// TIA Portal V20 export
FUNCTION "CollectAlarms" : Void   // FC61, LAD
TITLE = U1Em1_SepaUnwinderBottom
// stored: Namespace Unit1.Em1, SetENOAutomatically false
   VAR_INPUT
      resetAlarms : Bool;
      disableAlarms : Bool;
   END_VAR
   VAR_OUTPUT
      commandsToUnit : "LUC_typeStateCommands";   // Feedback to the unit
   END_VAR
   VAR CONSTANT
      DelayTime : Time := T#300ms;
      NoDelayTime : Time;
   END_VAR
BEGIN

REGION Network 1: Reset Alarms
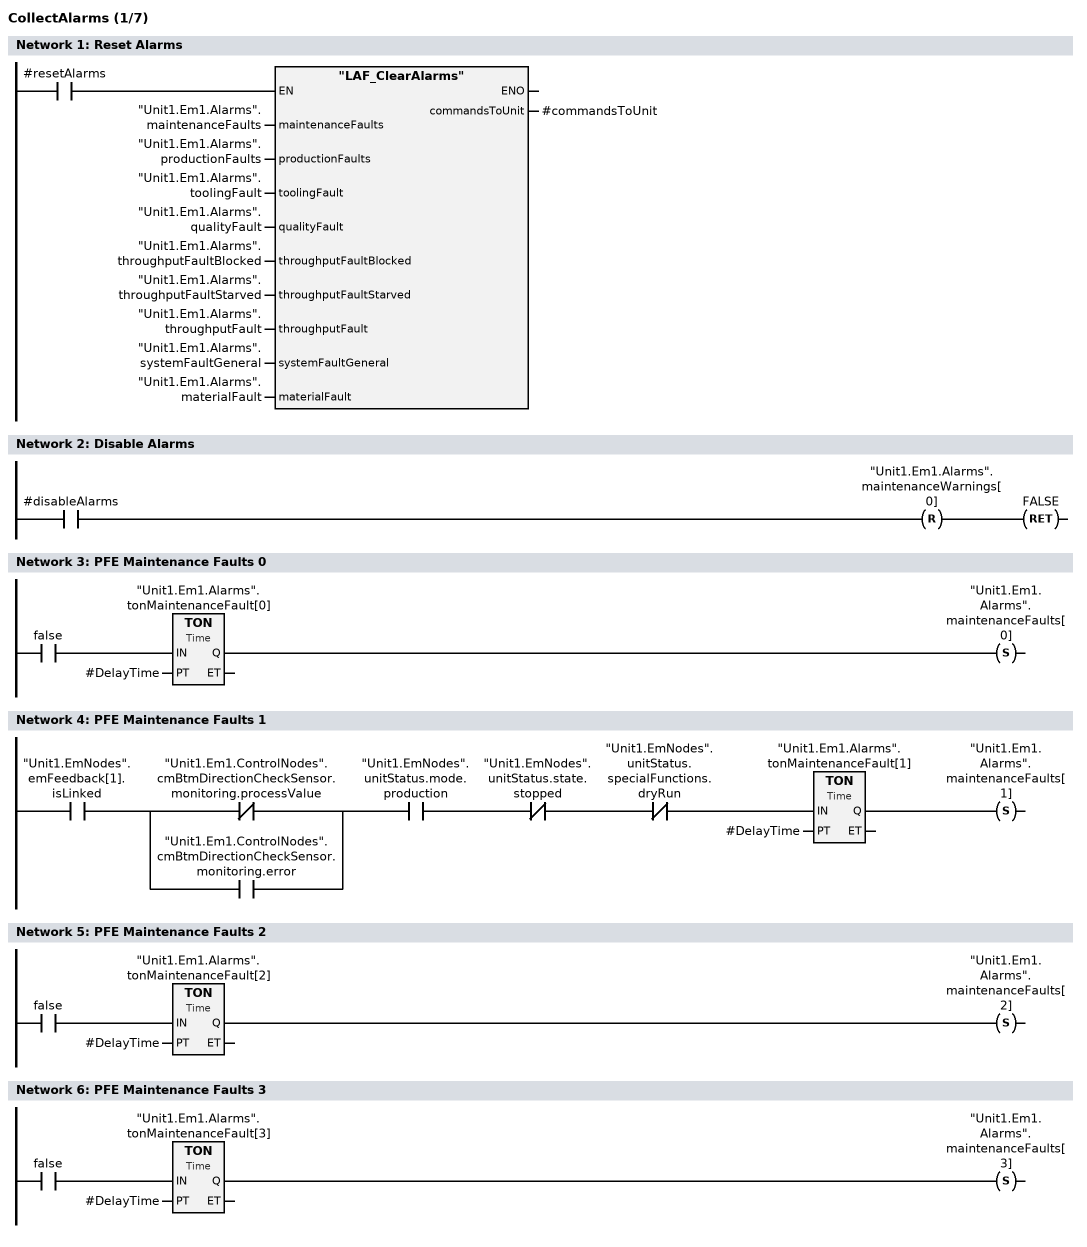
   RUNG wire#powerrail
      Contact( #resetAlarms )
      "LAF_ClearAlarms"(maintenanceFaults := "Unit1.Em1.Alarms".maintenanceFaults, productionFaults := "Unit1.Em1.Alarms".productionFaults, toolingFault := "Unit1.Em1.Alarms".toolingFault, qualityFault := "Unit1.Em1.Alarms".qualityFault, throughputFaultBlocked := "Unit1.Em1.Alarms".throughputFaultBlocked, throughputFaultStarved := "Unit1.Em1.Alarms".throughputFaultStarved, throughputFault := "Unit1.Em1.Alarms".throughputFault, systemFaultGeneral := "Unit1.Em1.Alarms".systemFaultGeneral, materialFault := "Unit1.Em1.Alarms".materialFault, commandsToUnit => #commandsToUnit)
   END_RUNG
   // the same network as SCL:
   IF #resetAlarms THEN
       "LAF_ClearAlarms"(maintenanceFaults := "Unit1.Em1.Alarms".maintenanceFaults,
                         productionFaults := "Unit1.Em1.Alarms".productionFaults,
                         toolingFault := "Unit1.Em1.Alarms".toolingFault,
                         qualityFault := "Unit1.Em1.Alarms".qualityFault,
                         throughputFaultBlocked := "Unit1.Em1.Alarms".throughputFaultBlocked,
                         throughputFaultStarved := "Unit1.Em1.Alarms".throughputFaultStarved,
                         throughputFault := "Unit1.Em1.Alarms".throughputFault,
                         systemFaultGeneral := "Unit1.Em1.Alarms".systemFaultGeneral,
                         materialFault := "Unit1.Em1.Alarms".materialFault,
                         commandsToUnit => #commandsToUnit);
   END_IF;
END_REGION

REGION Network 2: Disable Alarms
   RUNG wire#powerrail
      Contact( #disableAlarms )
      R_Coil( "Unit1.Em1.Alarms".maintenanceWarnings[0] )
      ReturnCoil( FALSE )
   END_RUNG
   // the same network as SCL:
   IF #disableAlarms THEN
       "Unit1.Em1.Alarms".maintenanceWarnings[0] := FALSE;
       ENO := FALSE;
       RETURN;
   END_IF;
END_REGION

REGION Network 3: PFE Maintenance Faults 0
   RUNG wire#powerrail
      Contact( false )
      { S7_Templates := "time_type := Time" } "Unit1.Em1.Alarms".tonMaintenanceFault[0].TON(pt := #DelayTime, et =>)
      S_Coil( "Unit1.Em1.Alarms".maintenanceFaults[0] )
   END_RUNG
   // the same network as SCL:
   "Unit1.Em1.Alarms".tonMaintenanceFault[0].TON(IN := false, PT := #DelayTime);
   IF "Unit1.Em1.Alarms".tonMaintenanceFault[0].Q THEN
       "Unit1.Em1.Alarms".maintenanceFaults[0] := TRUE;
   END_IF;
END_REGION

REGION Network 4: PFE Maintenance Faults 1
   RUNG wire#powerrail
      Contact( "Unit1.EmNodes".emFeedback[1].isLinked )
      wire#w1
      I_Contact( "Unit1.Em1.ControlNodes".cmBtmDirectionCheckSensor.monitoring.processValue )
      wire#w2
      Contact( "Unit1.EmNodes".unitStatus.mode.production )
      I_Contact( "Unit1.EmNodes".unitStatus.state.stopped )
      I_Contact( "Unit1.EmNodes".unitStatus.specialFunctions.dryRun )
      { S7_Templates := "time_type := Time" } "Unit1.Em1.Alarms".tonMaintenanceFault[1].TON(pt := #DelayTime, et =>)
      S_Coil( "Unit1.Em1.Alarms".maintenanceFaults[1] )
   END_RUNG
   RUNG wire#w1
      Contact( "Unit1.Em1.ControlNodes".cmBtmDirectionCheckSensor.monitoring.error )
   END_RUNG wire#w2
   // the same network as SCL:
   "Unit1.Em1.Alarms".tonMaintenanceFault[1].TON(IN := "Unit1.EmNodes".emFeedback[1].isLinked AND (NOT "Unit1.Em1.ControlNodes".cmBtmDirectionCheckSensor.monitoring.processValue OR "Unit1.Em1.ControlNodes".cmBtmDirectionCheckSensor.monitoring.error) AND "Unit1.EmNodes".unitStatus.mode.production AND NOT "Unit1.EmNodes".unitStatus.state.stopped AND NOT "Unit1.EmNodes".unitStatus.specialFunctions.dryRun,
                           PT := #DelayTime);
   IF "Unit1.Em1.Alarms".tonMaintenanceFault[1].Q THEN
       "Unit1.Em1.Alarms".maintenanceFaults[1] := TRUE;
   END_IF;
END_REGION

REGION Network 5: PFE Maintenance Faults 2
   RUNG wire#powerrail
      Contact( false )
      { S7_Templates := "time_type := Time" } "Unit1.Em1.Alarms".tonMaintenanceFault[2].TON(pt := #DelayTime, et =>)
      S_Coil( "Unit1.Em1.Alarms".maintenanceFaults[2] )
   END_RUNG
   // the same network as SCL:
   "Unit1.Em1.Alarms".tonMaintenanceFault[2].TON(IN := false, PT := #DelayTime);
   IF "Unit1.Em1.Alarms".tonMaintenanceFault[2].Q THEN
       "Unit1.Em1.Alarms".maintenanceFaults[2] := TRUE;
   END_IF;
END_REGION

REGION Network 6: PFE Maintenance Faults 3
   RUNG wire#powerrail
      Contact( false )
      { S7_Templates := "time_type := Time" } "Unit1.Em1.Alarms".tonMaintenanceFault[3].TON(pt := #DelayTime, et =>)
      S_Coil( "Unit1.Em1.Alarms".maintenanceFaults[3] )
   END_RUNG
   // the same network as SCL:
   "Unit1.Em1.Alarms".tonMaintenanceFault[3].TON(IN := false, PT := #DelayTime);
   IF "Unit1.Em1.Alarms".tonMaintenanceFault[3].Q THEN
       "Unit1.Em1.Alarms".maintenanceFaults[3] := TRUE;
   END_IF;
END_REGION

REGION Network 7: PFE Maintenance Faults 4
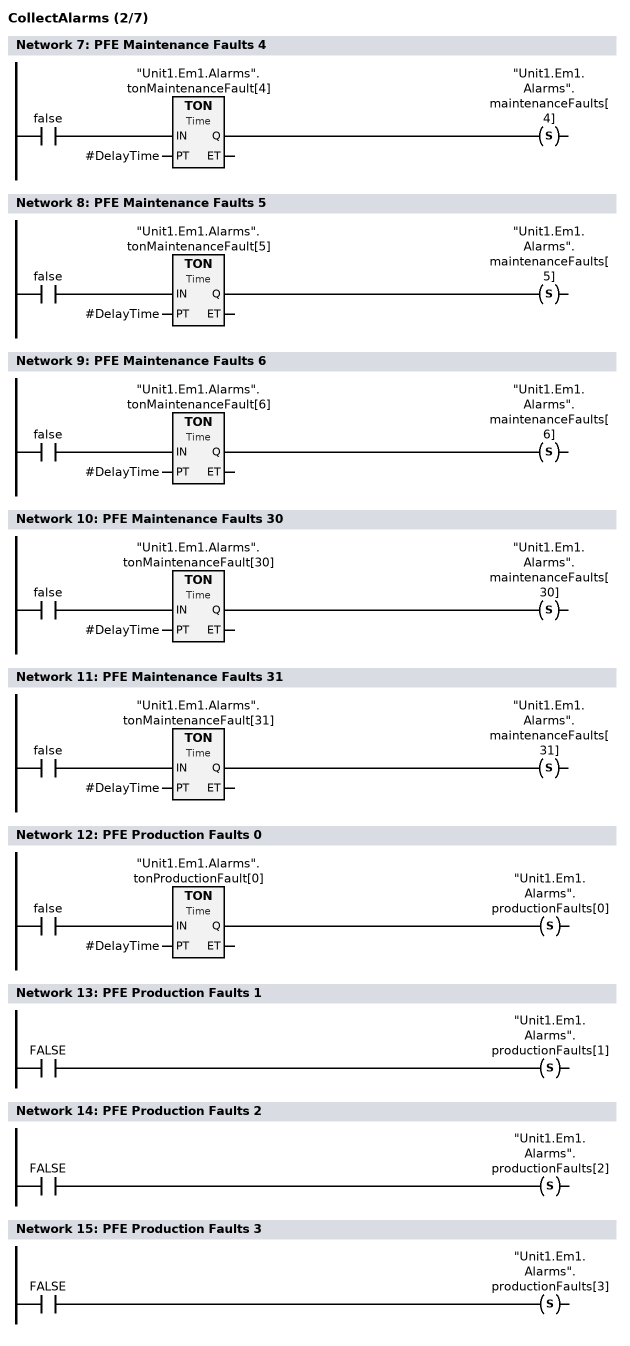
   RUNG wire#powerrail
      Contact( false )
      { S7_Templates := "time_type := Time" } "Unit1.Em1.Alarms".tonMaintenanceFault[4].TON(pt := #DelayTime, et =>)
      S_Coil( "Unit1.Em1.Alarms".maintenanceFaults[4] )
   END_RUNG
   // the same network as SCL:
   "Unit1.Em1.Alarms".tonMaintenanceFault[4].TON(IN := false, PT := #DelayTime);
   IF "Unit1.Em1.Alarms".tonMaintenanceFault[4].Q THEN
       "Unit1.Em1.Alarms".maintenanceFaults[4] := TRUE;
   END_IF;
END_REGION

REGION Network 8: PFE Maintenance Faults 5
   RUNG wire#powerrail
      Contact( false )
      { S7_Templates := "time_type := Time" } "Unit1.Em1.Alarms".tonMaintenanceFault[5].TON(pt := #DelayTime, et =>)
      S_Coil( "Unit1.Em1.Alarms".maintenanceFaults[5] )
   END_RUNG
   // the same network as SCL:
   "Unit1.Em1.Alarms".tonMaintenanceFault[5].TON(IN := false, PT := #DelayTime);
   IF "Unit1.Em1.Alarms".tonMaintenanceFault[5].Q THEN
       "Unit1.Em1.Alarms".maintenanceFaults[5] := TRUE;
   END_IF;
END_REGION

REGION Network 9: PFE Maintenance Faults 6
   RUNG wire#powerrail
      Contact( false )
      { S7_Templates := "time_type := Time" } "Unit1.Em1.Alarms".tonMaintenanceFault[6].TON(pt := #DelayTime, et =>)
      S_Coil( "Unit1.Em1.Alarms".maintenanceFaults[6] )
   END_RUNG
   // the same network as SCL:
   "Unit1.Em1.Alarms".tonMaintenanceFault[6].TON(IN := false, PT := #DelayTime);
   IF "Unit1.Em1.Alarms".tonMaintenanceFault[6].Q THEN
       "Unit1.Em1.Alarms".maintenanceFaults[6] := TRUE;
   END_IF;
END_REGION

REGION Network 10: PFE Maintenance Faults 30
   RUNG wire#powerrail
      Contact( false )
      { S7_Templates := "time_type := Time" } "Unit1.Em1.Alarms".tonMaintenanceFault[30].TON(pt := #DelayTime, et =>)
      S_Coil( "Unit1.Em1.Alarms".maintenanceFaults[30] )
   END_RUNG
   // the same network as SCL:
   "Unit1.Em1.Alarms".tonMaintenanceFault[30].TON(IN := false, PT := #DelayTime);
   IF "Unit1.Em1.Alarms".tonMaintenanceFault[30].Q THEN
       "Unit1.Em1.Alarms".maintenanceFaults[30] := TRUE;
   END_IF;
END_REGION

REGION Network 11: PFE Maintenance Faults 31
   RUNG wire#powerrail
      Contact( false )
      { S7_Templates := "time_type := Time" } "Unit1.Em1.Alarms".tonMaintenanceFault[31].TON(pt := #DelayTime, et =>)
      S_Coil( "Unit1.Em1.Alarms".maintenanceFaults[31] )
   END_RUNG
   // the same network as SCL:
   "Unit1.Em1.Alarms".tonMaintenanceFault[31].TON(IN := false, PT := #DelayTime);
   IF "Unit1.Em1.Alarms".tonMaintenanceFault[31].Q THEN
       "Unit1.Em1.Alarms".maintenanceFaults[31] := TRUE;
   END_IF;
END_REGION

REGION Network 12: PFE Production Faults 0
   RUNG wire#powerrail
      Contact( false )
      { S7_Templates := "time_type := Time" } "Unit1.Em1.Alarms".tonProductionFault[0].TON(pt := #DelayTime, et =>)
      S_Coil( "Unit1.Em1.Alarms".productionFaults[0] )
   END_RUNG
   // the same network as SCL:
   "Unit1.Em1.Alarms".tonProductionFault[0].TON(IN := false, PT := #DelayTime);
   IF "Unit1.Em1.Alarms".tonProductionFault[0].Q THEN "Unit1.Em1.Alarms".productionFaults[0] := TRUE; END_IF;
END_REGION

REGION Network 13: PFE Production Faults 1
   RUNG wire#powerrail
      Contact( FALSE )
      S_Coil( "Unit1.Em1.Alarms".productionFaults[1] )
   END_RUNG
   // the same network as SCL:
   IF FALSE THEN "Unit1.Em1.Alarms".productionFaults[1] := TRUE; END_IF;
END_REGION

REGION Network 14: PFE Production Faults 2
   RUNG wire#powerrail
      Contact( FALSE )
      S_Coil( "Unit1.Em1.Alarms".productionFaults[2] )
   END_RUNG
   // the same network as SCL:
   IF FALSE THEN "Unit1.Em1.Alarms".productionFaults[2] := TRUE; END_IF;
END_REGION

REGION Network 15: PFE Production Faults 3
   RUNG wire#powerrail
      Contact( FALSE )
      S_Coil( "Unit1.Em1.Alarms".productionFaults[3] )
   END_RUNG
   // the same network as SCL:
   IF FALSE THEN "Unit1.Em1.Alarms".productionFaults[3] := TRUE; END_IF;
END_REGION

REGION Network 16: PFE Production Faults 4
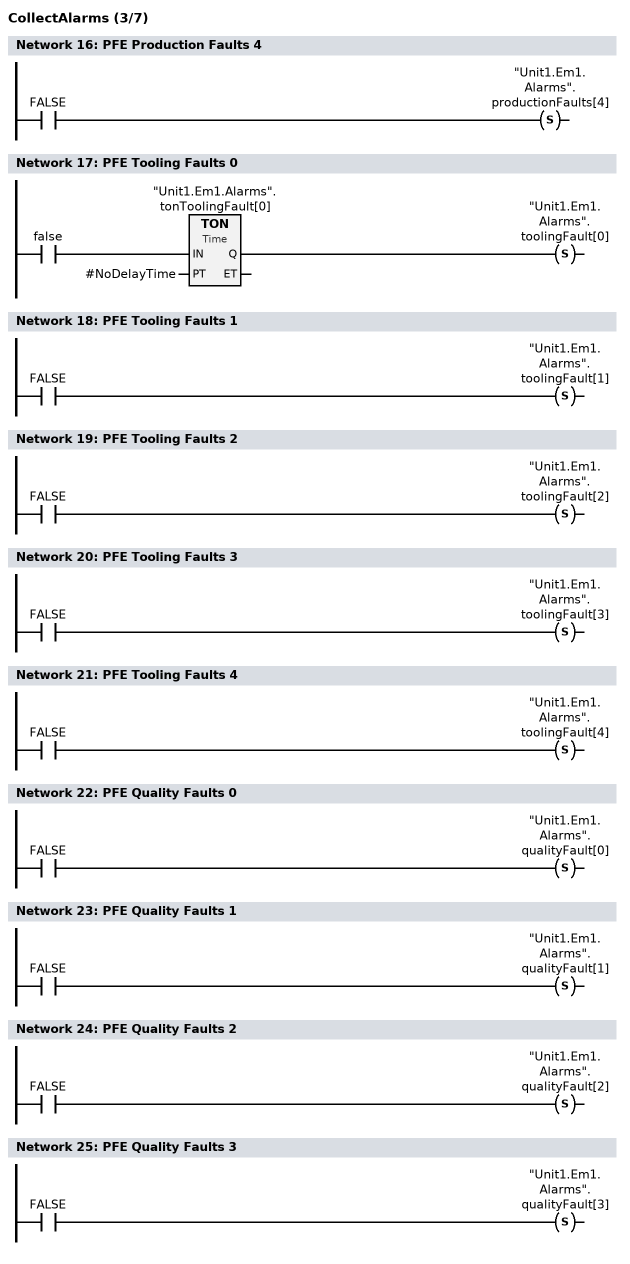
   RUNG wire#powerrail
      Contact( FALSE )
      S_Coil( "Unit1.Em1.Alarms".productionFaults[4] )
   END_RUNG
   // the same network as SCL:
   IF FALSE THEN "Unit1.Em1.Alarms".productionFaults[4] := TRUE; END_IF;
END_REGION

REGION Network 17: PFE Tooling Faults 0
   RUNG wire#powerrail
      Contact( false )
      { S7_Templates := "time_type := Time" } "Unit1.Em1.Alarms".tonToolingFault[0].TON(pt := #NoDelayTime, et =>)
      S_Coil( "Unit1.Em1.Alarms".toolingFault[0] )
   END_RUNG
   // the same network as SCL:
   "Unit1.Em1.Alarms".tonToolingFault[0].TON(IN := false, PT := #NoDelayTime);
   IF "Unit1.Em1.Alarms".tonToolingFault[0].Q THEN "Unit1.Em1.Alarms".toolingFault[0] := TRUE; END_IF;
END_REGION

REGION Network 18: PFE Tooling Faults 1
   RUNG wire#powerrail
      Contact( FALSE )
      S_Coil( "Unit1.Em1.Alarms".toolingFault[1] )
   END_RUNG
   // the same network as SCL:
   IF FALSE THEN "Unit1.Em1.Alarms".toolingFault[1] := TRUE; END_IF;
END_REGION

REGION Network 19: PFE Tooling Faults 2
   RUNG wire#powerrail
      Contact( FALSE )
      S_Coil( "Unit1.Em1.Alarms".toolingFault[2] )
   END_RUNG
   // the same network as SCL:
   IF FALSE THEN "Unit1.Em1.Alarms".toolingFault[2] := TRUE; END_IF;
END_REGION

REGION Network 20: PFE Tooling Faults 3
   RUNG wire#powerrail
      Contact( FALSE )
      S_Coil( "Unit1.Em1.Alarms".toolingFault[3] )
   END_RUNG
   // the same network as SCL:
   IF FALSE THEN "Unit1.Em1.Alarms".toolingFault[3] := TRUE; END_IF;
END_REGION

REGION Network 21: PFE Tooling Faults 4
   RUNG wire#powerrail
      Contact( FALSE )
      S_Coil( "Unit1.Em1.Alarms".toolingFault[4] )
   END_RUNG
   // the same network as SCL:
   IF FALSE THEN "Unit1.Em1.Alarms".toolingFault[4] := TRUE; END_IF;
END_REGION

REGION Network 22: PFE Quality Faults 0
   RUNG wire#powerrail
      Contact( FALSE )
      S_Coil( "Unit1.Em1.Alarms".qualityFault[0] )
   END_RUNG
   // the same network as SCL:
   IF FALSE THEN "Unit1.Em1.Alarms".qualityFault[0] := TRUE; END_IF;
END_REGION

REGION Network 23: PFE Quality Faults 1
   RUNG wire#powerrail
      Contact( FALSE )
      S_Coil( "Unit1.Em1.Alarms".qualityFault[1] )
   END_RUNG
   // the same network as SCL:
   IF FALSE THEN "Unit1.Em1.Alarms".qualityFault[1] := TRUE; END_IF;
END_REGION

REGION Network 24: PFE Quality Faults 2
   RUNG wire#powerrail
      Contact( FALSE )
      S_Coil( "Unit1.Em1.Alarms".qualityFault[2] )
   END_RUNG
   // the same network as SCL:
   IF FALSE THEN "Unit1.Em1.Alarms".qualityFault[2] := TRUE; END_IF;
END_REGION

REGION Network 25: PFE Quality Faults 3
   RUNG wire#powerrail
      Contact( FALSE )
      S_Coil( "Unit1.Em1.Alarms".qualityFault[3] )
   END_RUNG
   // the same network as SCL:
   IF FALSE THEN "Unit1.Em1.Alarms".qualityFault[3] := TRUE; END_IF;
END_REGION

REGION Network 26: PFE Quality Faults 4
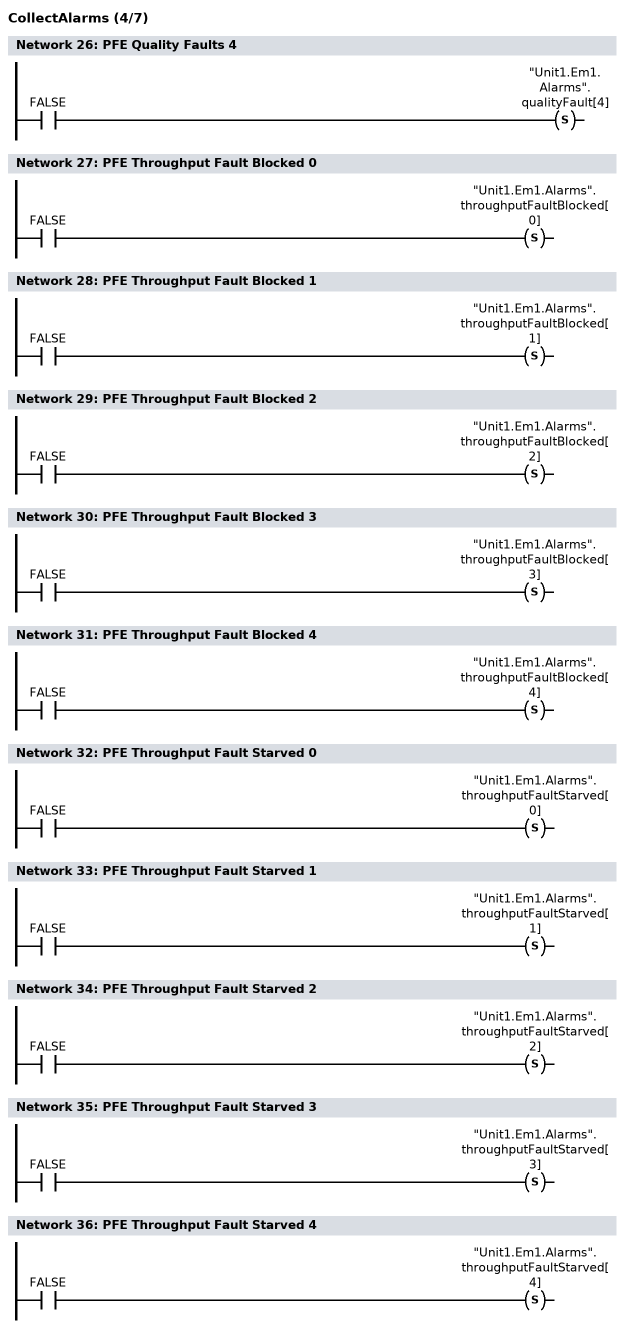
   RUNG wire#powerrail
      Contact( FALSE )
      S_Coil( "Unit1.Em1.Alarms".qualityFault[4] )
   END_RUNG
   // the same network as SCL:
   IF FALSE THEN "Unit1.Em1.Alarms".qualityFault[4] := TRUE; END_IF;
END_REGION

REGION Network 27: PFE Throughput Fault Blocked 0
   RUNG wire#powerrail
      Contact( FALSE )
      S_Coil( "Unit1.Em1.Alarms".throughputFaultBlocked[0] )
   END_RUNG
   // the same network as SCL:
   IF FALSE THEN "Unit1.Em1.Alarms".throughputFaultBlocked[0] := TRUE; END_IF;
END_REGION

REGION Network 28: PFE Throughput Fault Blocked 1
   RUNG wire#powerrail
      Contact( FALSE )
      S_Coil( "Unit1.Em1.Alarms".throughputFaultBlocked[1] )
   END_RUNG
   // the same network as SCL:
   IF FALSE THEN "Unit1.Em1.Alarms".throughputFaultBlocked[1] := TRUE; END_IF;
END_REGION

REGION Network 29: PFE Throughput Fault Blocked 2
   RUNG wire#powerrail
      Contact( FALSE )
      S_Coil( "Unit1.Em1.Alarms".throughputFaultBlocked[2] )
   END_RUNG
   // the same network as SCL:
   IF FALSE THEN "Unit1.Em1.Alarms".throughputFaultBlocked[2] := TRUE; END_IF;
END_REGION

REGION Network 30: PFE Throughput Fault Blocked 3
   RUNG wire#powerrail
      Contact( FALSE )
      S_Coil( "Unit1.Em1.Alarms".throughputFaultBlocked[3] )
   END_RUNG
   // the same network as SCL:
   IF FALSE THEN "Unit1.Em1.Alarms".throughputFaultBlocked[3] := TRUE; END_IF;
END_REGION

REGION Network 31: PFE Throughput Fault Blocked 4
   RUNG wire#powerrail
      Contact( FALSE )
      S_Coil( "Unit1.Em1.Alarms".throughputFaultBlocked[4] )
   END_RUNG
   // the same network as SCL:
   IF FALSE THEN "Unit1.Em1.Alarms".throughputFaultBlocked[4] := TRUE; END_IF;
END_REGION

REGION Network 32: PFE Throughput Fault Starved 0
   RUNG wire#powerrail
      Contact( FALSE )
      S_Coil( "Unit1.Em1.Alarms".throughputFaultStarved[0] )
   END_RUNG
   // the same network as SCL:
   IF FALSE THEN "Unit1.Em1.Alarms".throughputFaultStarved[0] := TRUE; END_IF;
END_REGION

REGION Network 33: PFE Throughput Fault Starved 1
   RUNG wire#powerrail
      Contact( FALSE )
      S_Coil( "Unit1.Em1.Alarms".throughputFaultStarved[1] )
   END_RUNG
   // the same network as SCL:
   IF FALSE THEN "Unit1.Em1.Alarms".throughputFaultStarved[1] := TRUE; END_IF;
END_REGION

REGION Network 34: PFE Throughput Fault Starved 2
   RUNG wire#powerrail
      Contact( FALSE )
      S_Coil( "Unit1.Em1.Alarms".throughputFaultStarved[2] )
   END_RUNG
   // the same network as SCL:
   IF FALSE THEN "Unit1.Em1.Alarms".throughputFaultStarved[2] := TRUE; END_IF;
END_REGION

REGION Network 35: PFE Throughput Fault Starved 3
   RUNG wire#powerrail
      Contact( FALSE )
      S_Coil( "Unit1.Em1.Alarms".throughputFaultStarved[3] )
   END_RUNG
   // the same network as SCL:
   IF FALSE THEN "Unit1.Em1.Alarms".throughputFaultStarved[3] := TRUE; END_IF;
END_REGION

REGION Network 36: PFE Throughput Fault Starved 4
   RUNG wire#powerrail
      Contact( FALSE )
      S_Coil( "Unit1.Em1.Alarms".throughputFaultStarved[4] )
   END_RUNG
   // the same network as SCL:
   IF FALSE THEN "Unit1.Em1.Alarms".throughputFaultStarved[4] := TRUE; END_IF;
END_REGION

REGION Network 37: PFE Throughput Fault 0
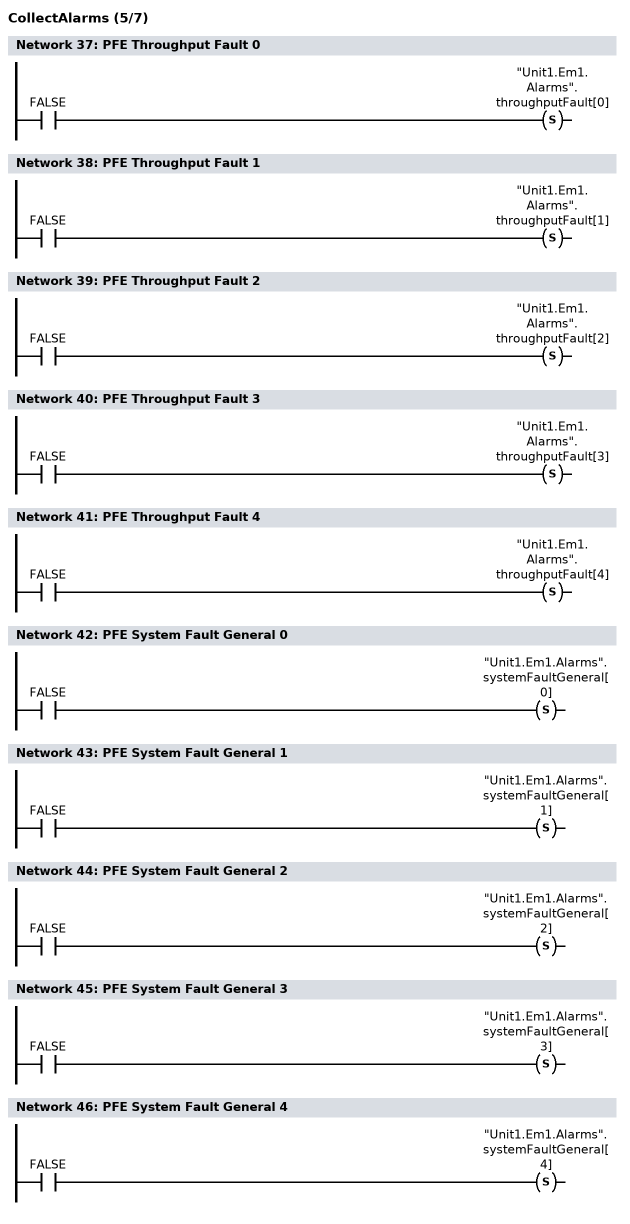
   RUNG wire#powerrail
      Contact( FALSE )
      S_Coil( "Unit1.Em1.Alarms".throughputFault[0] )
   END_RUNG
   // the same network as SCL:
   IF FALSE THEN "Unit1.Em1.Alarms".throughputFault[0] := TRUE; END_IF;
END_REGION

REGION Network 38: PFE Throughput Fault 1
   RUNG wire#powerrail
      Contact( FALSE )
      S_Coil( "Unit1.Em1.Alarms".throughputFault[1] )
   END_RUNG
   // the same network as SCL:
   IF FALSE THEN "Unit1.Em1.Alarms".throughputFault[1] := TRUE; END_IF;
END_REGION

REGION Network 39: PFE Throughput Fault 2
   RUNG wire#powerrail
      Contact( FALSE )
      S_Coil( "Unit1.Em1.Alarms".throughputFault[2] )
   END_RUNG
   // the same network as SCL:
   IF FALSE THEN "Unit1.Em1.Alarms".throughputFault[2] := TRUE; END_IF;
END_REGION

REGION Network 40: PFE Throughput Fault 3
   RUNG wire#powerrail
      Contact( FALSE )
      S_Coil( "Unit1.Em1.Alarms".throughputFault[3] )
   END_RUNG
   // the same network as SCL:
   IF FALSE THEN "Unit1.Em1.Alarms".throughputFault[3] := TRUE; END_IF;
END_REGION

REGION Network 41: PFE Throughput Fault 4
   RUNG wire#powerrail
      Contact( FALSE )
      S_Coil( "Unit1.Em1.Alarms".throughputFault[4] )
   END_RUNG
   // the same network as SCL:
   IF FALSE THEN "Unit1.Em1.Alarms".throughputFault[4] := TRUE; END_IF;
END_REGION

REGION Network 42: PFE System Fault General 0
   RUNG wire#powerrail
      Contact( FALSE )
      S_Coil( "Unit1.Em1.Alarms".systemFaultGeneral[0] )
   END_RUNG
   // the same network as SCL:
   IF FALSE THEN "Unit1.Em1.Alarms".systemFaultGeneral[0] := TRUE; END_IF;
END_REGION

REGION Network 43: PFE System Fault General 1
   RUNG wire#powerrail
      Contact( FALSE )
      S_Coil( "Unit1.Em1.Alarms".systemFaultGeneral[1] )
   END_RUNG
   // the same network as SCL:
   IF FALSE THEN "Unit1.Em1.Alarms".systemFaultGeneral[1] := TRUE; END_IF;
END_REGION

REGION Network 44: PFE System Fault General 2
   RUNG wire#powerrail
      Contact( FALSE )
      S_Coil( "Unit1.Em1.Alarms".systemFaultGeneral[2] )
   END_RUNG
   // the same network as SCL:
   IF FALSE THEN "Unit1.Em1.Alarms".systemFaultGeneral[2] := TRUE; END_IF;
END_REGION

REGION Network 45: PFE System Fault General 3
   RUNG wire#powerrail
      Contact( FALSE )
      S_Coil( "Unit1.Em1.Alarms".systemFaultGeneral[3] )
   END_RUNG
   // the same network as SCL:
   IF FALSE THEN "Unit1.Em1.Alarms".systemFaultGeneral[3] := TRUE; END_IF;
END_REGION

REGION Network 46: PFE System Fault General 4
   RUNG wire#powerrail
      Contact( FALSE )
      S_Coil( "Unit1.Em1.Alarms".systemFaultGeneral[4] )
   END_RUNG
   // the same network as SCL:
   IF FALSE THEN "Unit1.Em1.Alarms".systemFaultGeneral[4] := TRUE; END_IF;
END_REGION

REGION Network 47: PFE Material Fault 0
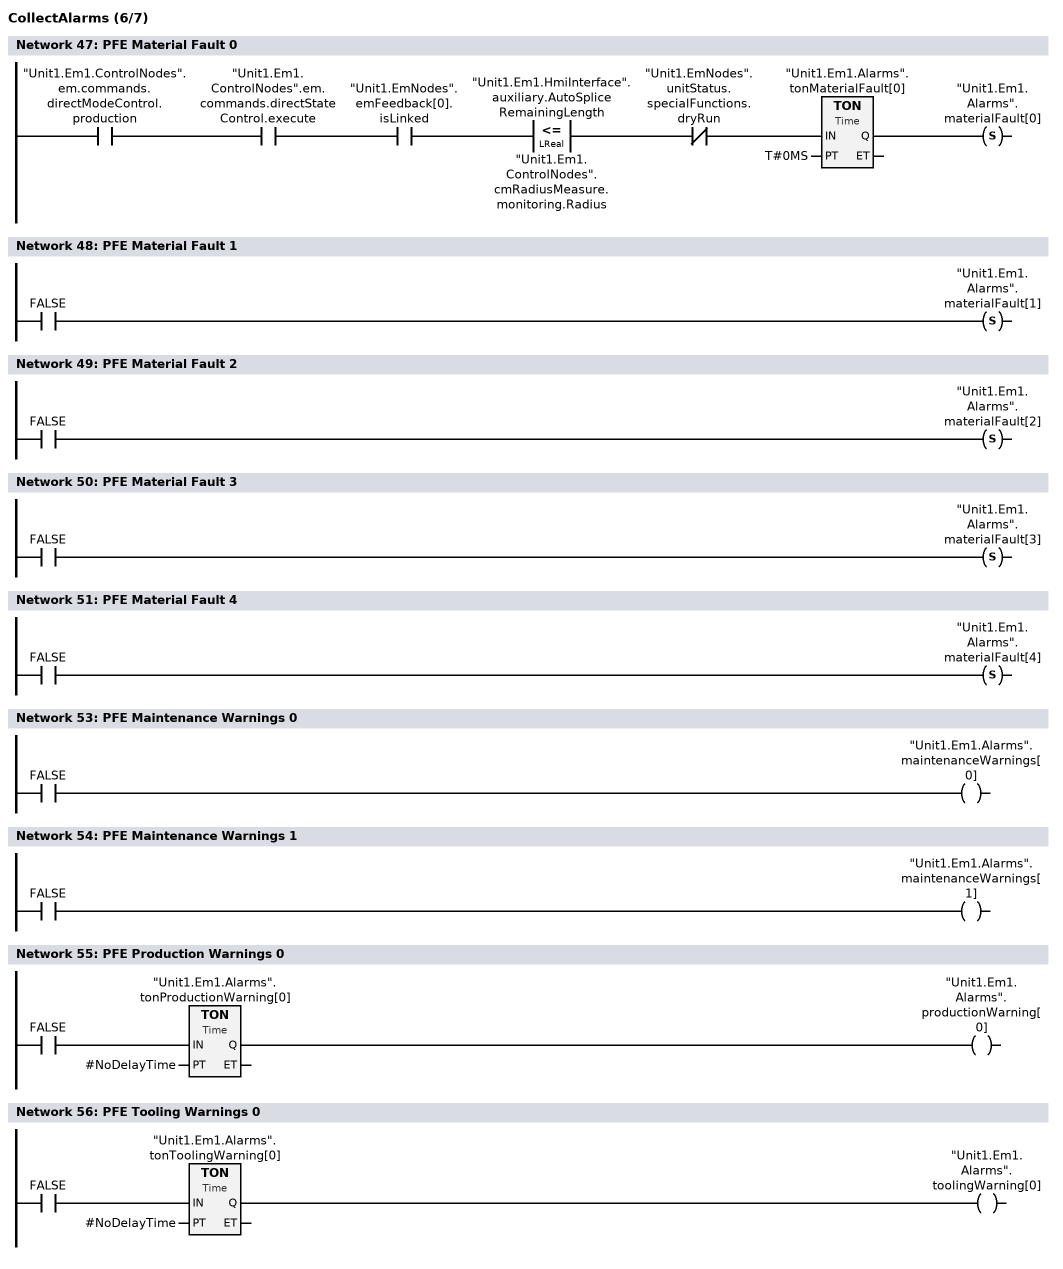
   RUNG wire#powerrail
      Contact( "Unit1.Em1.ControlNodes".em.commands.directModeControl.production )
      Contact( "Unit1.Em1.ControlNodes".em.commands.directStateControl.execute )
      Contact( "Unit1.EmNodes".emFeedback[0].isLinked )
      { S7_Templates := "SrcType := LReal" } LE_Contact(in1 := "Unit1.Em1.HmiInterface".auxiliary.AutoSpliceRemainingLength, in2 := "Unit1.Em1.ControlNodes".cmRadiusMeasure.monitoring.Radius)
      I_Contact( "Unit1.EmNodes".unitStatus.specialFunctions.dryRun )
      { S7_Templates := "time_type := Time" } "Unit1.Em1.Alarms".tonMaterialFault[0].TON(pt := T#0MS, et =>)
      S_Coil( "Unit1.Em1.Alarms".materialFault[0] )
   END_RUNG
   // the same network as SCL:
   "Unit1.Em1.Alarms".tonMaterialFault[0].TON(IN := "Unit1.Em1.ControlNodes".em.commands.directModeControl.production AND "Unit1.Em1.ControlNodes".em.commands.directStateControl.execute AND "Unit1.EmNodes".emFeedback[0].isLinked AND ("Unit1.Em1.HmiInterface".auxiliary.AutoSpliceRemainingLength <= "Unit1.Em1.ControlNodes".cmRadiusMeasure.monitoring.Radius) AND NOT "Unit1.EmNodes".unitStatus.specialFunctions.dryRun,
                           PT := T#0MS);
   IF "Unit1.Em1.Alarms".tonMaterialFault[0].Q THEN "Unit1.Em1.Alarms".materialFault[0] := TRUE; END_IF;
END_REGION

REGION Network 48: PFE Material Fault 1
   RUNG wire#powerrail
      Contact( FALSE )
      S_Coil( "Unit1.Em1.Alarms".materialFault[1] )
   END_RUNG
   // the same network as SCL:
   IF FALSE THEN "Unit1.Em1.Alarms".materialFault[1] := TRUE; END_IF;
END_REGION

REGION Network 49: PFE Material Fault 2
   RUNG wire#powerrail
      Contact( FALSE )
      S_Coil( "Unit1.Em1.Alarms".materialFault[2] )
   END_RUNG
   // the same network as SCL:
   IF FALSE THEN "Unit1.Em1.Alarms".materialFault[2] := TRUE; END_IF;
END_REGION

REGION Network 50: PFE Material Fault 3
   RUNG wire#powerrail
      Contact( FALSE )
      S_Coil( "Unit1.Em1.Alarms".materialFault[3] )
   END_RUNG
   // the same network as SCL:
   IF FALSE THEN "Unit1.Em1.Alarms".materialFault[3] := TRUE; END_IF;
END_REGION

REGION Network 51: PFE Material Fault 4
   RUNG wire#powerrail
      Contact( FALSE )
      S_Coil( "Unit1.Em1.Alarms".materialFault[4] )
   END_RUNG
   // the same network as SCL:
   IF FALSE THEN "Unit1.Em1.Alarms".materialFault[4] := TRUE; END_IF;
END_REGION

REGION Network 52: *************** Warning **************************
END_REGION

REGION Network 53: PFE Maintenance Warnings 0
   RUNG wire#powerrail
      Contact( FALSE )
      Coil( "Unit1.Em1.Alarms".maintenanceWarnings[0] )
   END_RUNG
   // the same network as SCL:
   "Unit1.Em1.Alarms".maintenanceWarnings[0] := FALSE;
END_REGION

REGION Network 54: PFE Maintenance Warnings 1
   RUNG wire#powerrail
      Contact( FALSE )
      Coil( "Unit1.Em1.Alarms".maintenanceWarnings[1] )
   END_RUNG
   // the same network as SCL:
   "Unit1.Em1.Alarms".maintenanceWarnings[1] := FALSE;
END_REGION

REGION Network 55: PFE Production Warnings 0
   RUNG wire#powerrail
      Contact( FALSE )
      { S7_Templates := "time_type := Time" } "Unit1.Em1.Alarms".tonProductionWarning[0].TON(pt := #NoDelayTime, et =>)
      Coil( "Unit1.Em1.Alarms".productionWarning[0] )
   END_RUNG
   // the same network as SCL:
   "Unit1.Em1.Alarms".tonProductionWarning[0].TON(IN := FALSE, PT := #NoDelayTime);
   "Unit1.Em1.Alarms".productionWarning[0] := "Unit1.Em1.Alarms".tonProductionWarning[0].Q;
END_REGION

REGION Network 56: PFE Tooling Warnings 0
   RUNG wire#powerrail
      Contact( FALSE )
      { S7_Templates := "time_type := Time" } "Unit1.Em1.Alarms".tonToolingWarning[0].TON(pt := #NoDelayTime, et =>)
      Coil( "Unit1.Em1.Alarms".toolingWarning[0] )
   END_RUNG
   // the same network as SCL:
   "Unit1.Em1.Alarms".tonToolingWarning[0].TON(IN := FALSE, PT := #NoDelayTime);
   "Unit1.Em1.Alarms".toolingWarning[0] := "Unit1.Em1.Alarms".tonToolingWarning[0].Q;
END_REGION

REGION Network 57: *************** Status ***************************
END_REGION

REGION Network 58: PFE Maintenance Status 0
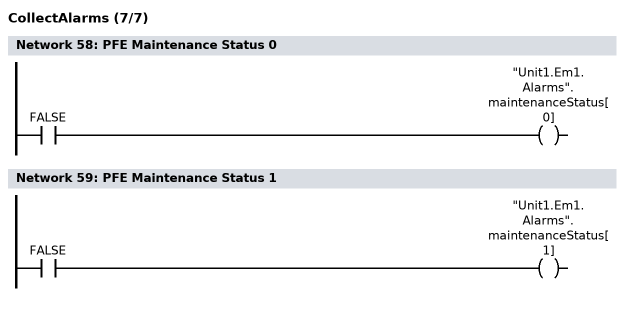
   RUNG wire#powerrail
      Contact( FALSE )
      Coil( "Unit1.Em1.Alarms".maintenanceStatus[0] )
   END_RUNG
   // the same network as SCL:
   "Unit1.Em1.Alarms".maintenanceStatus[0] := FALSE;
END_REGION

REGION Network 59: PFE Maintenance Status 1
   RUNG wire#powerrail
      Contact( FALSE )
      Coil( "Unit1.Em1.Alarms".maintenanceStatus[1] )
   END_RUNG
   // the same network as SCL:
   "Unit1.Em1.Alarms".maintenanceStatus[1] := FALSE;
END_REGION
END_FUNCTION
